(* IEC 61131-3 sources: Industry-PLC-LLM/data/PLCBEAD_repo/PLCBEAD_PLCEmbed-main/PLC-BEAD/Source/GEB/SETUP_EXTENDED_ASCII, 1 file *)

(* ---- SETUP_EXTENDED_ASCII.ST ---- *)
FUNCTION SETUP_EXTENDED_ASCII:BOOL

	VAR_INPUT
		X :	BOOL;
	END_VAR

	SETUP_EXTENDED_ASCII := X OR TRUE;
END_FUNCTION

PROGRAM program0
  VAR
	X :	BOOL;
    CEIL5_OUT : BOOL;
  END_VAR

  CEIL5_OUT := SETUP_EXTENDED_ASCII(X);
END_PROGRAM
